/// Concrete logger that dispatches to the process-global `LogManager` singleton.
///
/// Declare one instance per component/axis/subsystem and pass `name` to
/// `FB_Init` — the name becomes the `source` field on every log record so
/// you can filter by component in your log viewer.
///
/// Simple usage:
/// ```st
/// VAR
///   log : DefaultLogger('AxisX');
/// END_VAR
/// log.Info('Homing started');
/// log.Error('Limit switch triggered');
/// ```
///
/// Structured attributes and conditional logging:
/// ```st
/// log.WithAttribute('state', 'Homing').WithAttribute('speed', '100').Info('Axis moving');
/// log.OnCondition(error_active).Error('Drive fault detected');
/// ```
///
/// No wiring required — `FB_Init` connects automatically to `GetLogManager()`.
/// Register appenders on `GetLogManager()` once at program startup.
{attribute 'linkalways'}
{attribute 'no_explicit_call' := 'This FB is a CLASS and must be accessed using methods or properties'}
{attribute 'enable_dynamic_creation'}
{attribute 'reflection'}
FUNCTION_BLOCK PUBLIC DefaultLogger IMPLEMENTS Logger
VAR
	{attribute 'instance-path'}
    {attribute 'noinit'}
    instance_path : STRING(255);
	
	_name : STRING(255);
	attributes : ARRAY[0..9] OF LogAttribute;
	attribute_count : USINT;
	condition : BOOL := TRUE;
	chain_started : BOOL;
END_VAR
VAR CONSTANT
	INSTANCE_PATH_KEY_NAME : STRING := 'instance_path';
END_VAR

/// Log at DEBUG level.
METHOD PUBLIC Debug : BOOL
VAR_INPUT
	message : Tc2_System.T_MaxString;
END_VAR
InitChain();
IF condition THEN
	GetLogManager().Dispatch(LogLevel.Debug, message, _name, attributes, attribute_count);
END_IF
ResetChain();
Debug := TRUE;
END_METHOD

/// Log at ERROR level.
METHOD PUBLIC Error : BOOL
VAR_INPUT
	message : Tc2_System.T_MaxString;
END_VAR
InitChain();
IF condition THEN
	GetLogManager().Dispatch(LogLevel.Error, message, _name, attributes, attribute_count);
END_IF
ResetChain();
Error := TRUE;
END_METHOD

/// Log at FATAL level.
METHOD PUBLIC Fatal : BOOL
VAR_INPUT
	message : Tc2_System.T_MaxString;
END_VAR
InitChain();
IF condition THEN
	GetLogManager().Dispatch(LogLevel.Fatal, message, _name, attributes, attribute_count);
END_IF
ResetChain();
Fatal := TRUE;
END_METHOD

METHOD FB_Init : BOOL
VAR_INPUT
	bInitRetains : BOOL;
	bInCopyCode : BOOL;
	/// Component name used as the `source` field on every log record.
	name : STRING(63);
END_VAR
_name := name;
END_METHOD

/// Log at INFORMATION level.
METHOD PUBLIC Info : BOOL
VAR_INPUT
	message : Tc2_System.T_MaxString;
END_VAR
InitChain();
IF condition THEN
	GetLogManager().Dispatch(LogLevel.Information, message, _name, attributes, attribute_count);
END_IF
ResetChain();
Info := TRUE;
END_METHOD

// Initialise chain state on the first call of a log chain.
// Idempotent — safe to call from every chain method.
{attribute 'hide'}
METHOD PRIVATE InitChain
IF NOT chain_started THEN
	chain_started := TRUE;
	condition := TRUE;
	attribute_count := 0;
END_IF
END_METHOD

/// Component name used as the `source` field on every log record.
{attribute 'monitoring' := 'call'}
PROPERTY PUBLIC Name : STRING(63)
GET // PUBLIC
Name := _name;
END_GET
SET // PUBLIC
_name := Name;
END_SET
END_PROPERTY

/// Conditionally emit the log record.
/// When `cond` is FALSE the chain is still initialised but the terminal
/// method (`Debug`, `Info`, etc.) will be a no-op.
/// ```st
/// log.OnCondition(error_active).Error('Drive fault');
/// ```
METHOD PUBLIC OnCondition : REFERENCE TO DefaultLogger
VAR_INPUT
	cond : BOOL;
END_VAR
InitChain();
condition := cond;
OnCondition REF= THIS^;
END_METHOD

// Reset chain state after a terminal method completes.
// Must be called at the end of every Debug/Info/Warning/Error/Fatal implementation.
{attribute 'hide'}
METHOD PRIVATE ResetChain
chain_started := FALSE;
condition := TRUE;
attribute_count := 0;
END_METHOD

/// Log at WARNING level.
METHOD PUBLIC Warning : BOOL
VAR_INPUT
	message : Tc2_System.T_MaxString;
END_VAR
InitChain();
IF condition THEN
	GetLogManager().Dispatch(LogLevel.Warning, message, _name, attributes, attribute_count);
END_IF
ResetChain();
Warning := TRUE;
END_METHOD

/// Attach a string key/value attribute to the current log record.
/// Call before the terminal method (`Debug`, `Info`, `Warning`, `Error`, `Fatal`).
/// Up to 10 attributes per record; extras are silently ignored.
/// Chainable:
/// ```st
/// log.WithAttribute('state', 'Homing').WithDIntAttribute('pos', position).Info('Moving');
/// ```
METHOD PUBLIC WithAttribute : REFERENCE TO DefaultLogger
VAR_INPUT
	key : STRING(31);
	value : STRING(62);
END_VAR
InitChain();

IF attribute_count < 10 THEN
	attributes[attribute_count].key := key;
	attributes[attribute_count].attr_type := LogAttributeType.Str;
	Tc2_System.MemCpy(ADR(attributes[attribute_count].value_bytes[0]), ADR(value), SIZEOF(STRING(62)));
	attribute_count := attribute_count + 1;
END_IF

WithAttribute REF= THIS^;
END_METHOD

/// Attach a BOOL attribute.
METHOD PUBLIC WithBoolAttribute : REFERENCE TO DefaultLogger
VAR_INPUT
	key : STRING(31);
	value : BOOL;
END_VAR
InitChain();

IF attribute_count < 10 THEN
	attributes[attribute_count].key := key;
	attributes[attribute_count].attr_type := LogAttributeType.Boolean;
	attributes[attribute_count].value_bytes[0] := BOOL_TO_BYTE(value);
	attribute_count := attribute_count + 1;
END_IF

WithBoolAttribute REF= THIS^;
END_METHOD

/// Attach a DINT (32-bit signed) attribute.
METHOD PUBLIC WithDIntAttribute : REFERENCE TO DefaultLogger
VAR_INPUT
	key : STRING(31);
	value : DINT;
END_VAR
InitChain();

IF attribute_count < 10 THEN
	attributes[attribute_count].key := key;
	attributes[attribute_count].attr_type := LogAttributeType.Int32;
	Tc2_System.MemCpy(ADR(attributes[attribute_count].value_bytes[0]), ADR(value), SIZEOF(DINT));
	attribute_count := attribute_count + 1;
END_IF

WithDIntAttribute REF= THIS^;
END_METHOD

/// Attach the instance path to the current log record.
/// Call before the terminal method (`Debug`, `Info`, `Warning`, `Error`, `Fatal`).
/// Chainable:
/// ```st
/// log.WithInstancePath().WithDIntAttribute('pos', position).Info('Moving');
/// ```
METHOD PUBLIC WithInstancePath : REFERENCE TO DefaultLogger
WithInstancePath REF= WithAttribute(INSTANCE_PATH_KEY_NAME, instance_path);
END_METHOD

/// Attach an INT (16-bit signed) attribute.
METHOD PUBLIC WithIntAttribute : REFERENCE TO DefaultLogger
VAR_INPUT
	key : STRING(31);
	value : INT;
END_VAR
InitChain();

IF attribute_count < 10 THEN
	attributes[attribute_count].key := key;
	attributes[attribute_count].attr_type := LogAttributeType.Int16;
	Tc2_System.MemCpy(ADR(attributes[attribute_count].value_bytes[0]), ADR(value), SIZEOF(INT));
	attribute_count := attribute_count + 1;
END_IF

WithIntAttribute REF= THIS^;
END_METHOD

/// Attach a LINT (64-bit signed) attribute.
METHOD PUBLIC WithLIntAttribute : REFERENCE TO DefaultLogger
VAR_INPUT
	key : STRING(31);
	value : LINT;
END_VAR
InitChain();

IF attribute_count < 10 THEN
	attributes[attribute_count].key := key;
	attributes[attribute_count].attr_type := LogAttributeType.Int64;
	Tc2_System.MemCpy(ADR(attributes[attribute_count].value_bytes[0]), ADR(value), SIZEOF(LINT));
	attribute_count := attribute_count + 1;
END_IF

WithLIntAttribute REF= THIS^;
END_METHOD

/// Attach an LREAL (64-bit float) attribute.
METHOD PUBLIC WithLRealAttribute : REFERENCE TO DefaultLogger
VAR_INPUT
	key : STRING(31);
	value : LREAL;
END_VAR
InitChain();

IF attribute_count < 10 THEN
	attributes[attribute_count].key := key;
	attributes[attribute_count].attr_type := LogAttributeType.Float64;
	Tc2_System.MemCpy(ADR(attributes[attribute_count].value_bytes[0]), ADR(value), SIZEOF(LREAL));
	attribute_count := attribute_count + 1;
END_IF

WithLRealAttribute REF= THIS^;
END_METHOD

/// Attach a REAL (32-bit float) attribute.
METHOD PUBLIC WithRealAttribute : REFERENCE TO DefaultLogger
VAR_INPUT
	key : STRING(31);
	value : REAL;
END_VAR
InitChain();

IF attribute_count < 10 THEN
	attributes[attribute_count].key := key;
	attributes[attribute_count].attr_type := LogAttributeType.Float32;
	Tc2_System.MemCpy(ADR(attributes[attribute_count].value_bytes[0]), ADR(value), SIZEOF(REAL));
	attribute_count := attribute_count + 1;
END_IF

WithRealAttribute REF= THIS^;
END_METHOD

/// Attach a UDINT (32-bit unsigned) attribute.
METHOD PUBLIC WithUDIntAttribute : REFERENCE TO DefaultLogger
VAR_INPUT
	key : STRING(31);
	value : UDINT;
END_VAR
InitChain();

IF attribute_count < 10 THEN
	attributes[attribute_count].key := key;
	attributes[attribute_count].attr_type := LogAttributeType.Uint32;
	Tc2_System.MemCpy(ADR(attributes[attribute_count].value_bytes[0]), ADR(value), SIZEOF(UDINT));
	attribute_count := attribute_count + 1;
END_IF

WithUDIntAttribute REF= THIS^;
END_METHOD

/// Attach a UINT (16-bit unsigned) attribute.
METHOD PUBLIC WithUIntAttribute : REFERENCE TO DefaultLogger
VAR_INPUT
	key : STRING(31);
	value : UINT;
END_VAR
InitChain();

IF attribute_count < 10 THEN
	attributes[attribute_count].key := key;
	attributes[attribute_count].attr_type := LogAttributeType.Uint16;
	Tc2_System.MemCpy(ADR(attributes[attribute_count].value_bytes[0]), ADR(value), SIZEOF(UINT));
	attribute_count := attribute_count + 1;
END_IF

WithUIntAttribute REF= THIS^;
END_METHOD

/// Attach a ULINT (64-bit unsigned) attribute.
METHOD PUBLIC WithULIntAttribute : REFERENCE TO DefaultLogger
VAR_INPUT
	key : STRING(31);
	value : ULINT;
END_VAR
InitChain();

IF attribute_count < 10 THEN
	attributes[attribute_count].key := key;
	attributes[attribute_count].attr_type := LogAttributeType.Uint64;
	Tc2_System.MemCpy(ADR(attributes[attribute_count].value_bytes[0]), ADR(value), SIZEOF(ULINT));
	attribute_count := attribute_count + 1;
END_IF

WithULIntAttribute REF= THIS^;
END_METHOD

END_FUNCTION_BLOCK

(* stored: Version 1.1.0.1
   POU DefaultLogger: Id {1a2b3c4d-5e6f-7890-1a2b-3c4d5e6f7890}, SpecialFunc None
   Method Debug: Id {3c4d5e6f-7a8b-9012-3c4d-5e6f7a8b9012}
   Method Error: Id {6f7a8b9c-0d1e-2345-6f7a-8b9c0d1e2345}
   Method Fatal: Id {7a8b9c0d-1e2f-3456-7a8b-9c0d1e2f3456}
   Method FB_Init: Id {2b3c4d5e-6f7a-8901-2b3c-4d5e6f7a8901}
   Method Info: Id {4d5e6f7a-8b9c-0123-4d5e-6f7a8b9c0123}
   Method InitChain: Id {0d1e2f3a-4b5c-6789-0d1e-2f3a4b5c6789}
   Property Name: Id {2f3a4b5c-6d7e-8901-2f3a-4b5c6d7e8901}
   Get Get: Id {3a4b5c6d-7e8f-9012-3a4b-5c6d7e8f9012}
   Set Set: Id {4b5c6d7e-8f9a-0123-4b5c-6d7e8f9a0123}
   Method OnCondition: Id {9c0d1e2f-3a4b-5678-9c0d-1e2f3a4b5678}
   Method ResetChain: Id {1e2f3a4b-5c6d-7890-1e2f-3a4b5c6d7890}
   Method Warning: Id {5e6f7a8b-9c0d-1234-5e6f-7a8b9c0d1234}
   Method WithAttribute: Id {8b9c0d1e-2f3a-4567-8b9c-0d1e2f3a4567}
   Method WithBoolAttribute: Id {1a2b3c4d-5e6f-7001-1a2b-3c4d5e6f7001}
   Method WithDIntAttribute: Id {3c4d5e6f-7001-2233-3c4d-5e6f70012233}
   Method WithInstancePath: Id {62217dc2-2346-4aa1-8b58-8fd13aabdf15}
   Method WithIntAttribute: Id {2b3c4d5e-6f70-1122-2b3c-4d5e6f701122}
   Method WithLIntAttribute: Id {4d5e6f70-0112-3344-4d5e-6f7001123344}
   Method WithLRealAttribute: Id {12233445-5667-8899-1223-344556678899}
   Method WithRealAttribute: Id {01122334-4556-7788-0112-233445567788}
   Method WithUDIntAttribute: Id {6f700112-2334-5566-6f70-011223345566}
   Method WithUIntAttribute: Id {5e6f7001-1223-4455-5e6f-700112234455}
   Method WithULIntAttribute: Id {70011223-3445-6677-7001-122334456677} *)
